// TIA Portal V17 export
// export: Created 2024-08-26T21:07:18.828112Z, ExportSetting WithDefaults, DisplayName Totally Integrated Automation Portal, DisplayVersion V17 Update 7, DisplayName TIA Portal Openness, DisplayVersion V17 Update 7, DisplayName TIA Portal Version Control Interface, DisplayVersion V17, DisplayName SINAMICS Startdrive Advanced, DisplayVersion V17 SP2, DisplayName SINAMICS Startdrive G110M, G120, G120C, G120D, G120P, G115D, DisplayVersion V17 SP2, DisplayName SINAMICS Startdrive G130, G150, S120, S150, SINAMICS MV, S210, DisplayVersion V17 SP2, DisplayName STEP 7 Professional, DisplayVersion V17 Update 7, DisplayName STEP 7 Safety, DisplayVersion V17 Update 6, DisplayName WinCC Advanced / Unified PC, DisplayVersion V17 Update 7
DATA_BLOCK "sensorDistribution"   // DB129
{ S7_Optimized_Access := 'TRUE' }
VERSION : 0.1
// stored: AutoNumber false, DBAccessibleFromOPCUA true, DBAccessibleFromWebserver true, IsOnlyStoredInLoadMemory false, IsRetainMemResEnabled false, IsWriteProtectedInAS false, MemoryReserve 100
   VAR
      inputsStatus : Array[0..31] of Byte;
      outputsStatus : Array[0..31] of Byte;
   END_VAR
BEGIN
   inputsStatus[0..1] := 16#00;
   inputsStatus[2] := 16#01;
   inputsStatus[3..7] := 16#00;
   inputsStatus[8..9] := 16#01;
   inputsStatus[10] := 16#00;
   inputsStatus[11..13] := 16#01;
   inputsStatus[14..16] := 16#00;
   inputsStatus[17..18] := 16#01;
   inputsStatus[19..23] := 16#00;
   inputsStatus[24] := 16#01;
   inputsStatus[25..30] := 16#00;
   inputsStatus[31] := 16#01;
   outputsStatus[0] := 16#00;
   outputsStatus[1] := 16#01;
   outputsStatus[2] := 16#00;
   outputsStatus[3] := 16#01;
   outputsStatus[4] := 16#00;
   outputsStatus[5] := 16#01;
   outputsStatus[6] := 16#00;
   outputsStatus[7] := 16#01;
   outputsStatus[8..12] := 16#00;
   outputsStatus[13] := 16#01;
   outputsStatus[14..31] := 16#00;
END_DATA_BLOCK
